{attribute 'linkalways'} 
{attribute 'no_explicit_call' := 'This FB is a CLASS and must be accessed using methods or properties'}
{attribute 'enable_dynamic_creation'}
FUNCTION_BLOCK _ETcVnFeatureScoreTypeORB EXTENDS EnumDatatypeBase
VAR
	localData : ETcVnFeatureScoreTypeORB;
	activeData : REFERENCE TO ETcVnFeatureScoreTypeORB;
	enumBaseDatatype : _DINT(localData);
END_VAR

METHOD PRIVATE AddLocalEnumeration
VAR_INPUT
	Enumeration : T_MAXSTRING;
	Value : ETcVnFeatureScoreTypeORB;
END_VAR
AddEnumeration(Enumeration, Value);
END_METHOD

PROPERTY PUBLIC Address : PVOID
GET
Address := ADR(activeData);
END_GET
END_PROPERTY

METHOD PUBLIC ClearReference
VAR_INPUT
END_VAR
activeData REF= localData;
SetBaseDatatypeReference();
END_METHOD

METHOD PUBLIC Clone : I_Datatype
VAR
    pClone : POINTER TO _ETcVnFeatureScoreTypeORB;
END_VAR
pClone := __NEW(_ETcVnFeatureScoreTypeORB(InitialValue := Value));
Clone := pClone^;
END_METHOD

METHOD FB_init : BOOL
VAR_INPUT
	bInitRetains : BOOL; // if TRUE, the retain variables are initialized (warm start / cold start)
	bInCopyCode : BOOL;  // if TRUE, the instance afterwards gets moved into the copy code (online change)
	InitialValue : ETcVnFeatureScoreTypeORB;
END_VAR
localData := InitialValue;
AddBaseDatatype(enumBaseDatatype);
ClearReference();

AddLocalEnumeration('TCVN_FST_ORB_HARRIS', ETcVnFeatureScoreTypeORB.TCVN_FST_ORB_HARRIS);
AddLocalEnumeration('TCVN_FST_ORB_FAST', ETcVnFeatureScoreTypeORB.TCVN_FST_ORB_FAST);
END_METHOD

PROPERTY PUBLIC Identifier : T_MAXSTRING
GET
Identifier := 'ETcVnFeatureScoreTypeORB';
END_GET
END_PROPERTY

METHOD IsEnumeratorValueEqual : BOOL
VAR_INPUT
	Enumerator : I_KeyValueForwardEnumerator;
END_VAR
VAR
	storedValue : ETcVnFeatureScoreTypeORB;
END_VAR
IF NOT Enumerator.TryGet(storedValue) THEN
	RETURN;
END_IF

IsEnumeratorValueEqual := storedValue = activeData;
END_METHOD

METHOD PUBLIC MakeReferenceTo
VAR_INPUT
	ReferenceTarget : REFERENCE TO ETcVnFeatureScoreTypeORB;
END_VAR
activeData REF= ReferenceTarget;
SetBaseDatatypeReference();
END_METHOD

METHOD PROTECTED SetBaseDatatypeReference
VAR_INPUT
END_VAR
enumBaseDatatype.MakeReferenceTo(activeData);
END_METHOD

PROPERTY PUBLIC Size : UDINT
GET
Size := SIZEOF(activeData);
END_GET
END_PROPERTY

METHOD TryMakeReferenceTo : BOOL
VAR_INPUT
	Target : I_Datatype;
END_VAR
VAR
	targetAsEnum : I_EnumDatatype;
	pTargetData : POINTER TO ETcVnFeatureScoreTypeORB;
END_VAR
IF NOT Target.TryResolveAsEnumDatatype(targetAsEnum) THEN
	RETURN;
END_IF

IF targetAsEnum.Identifier <> Identifier THEN
	RETURN;
END_IF

pTargetData := Target.Address;
activeData REF= pTargetData^;
SetBaseDatatypeReference();
TryMakeReferenceTo := TRUE;
END_METHOD

PROPERTY PUBLIC Value : ETcVnFeatureScoreTypeORB
GET
Value := activeData;
END_GET
SET
activeData := Value;
END_SET
END_PROPERTY

END_FUNCTION_BLOCK

(* stored: Version 1.1.0.1
   POU _ETcVnFeatureScoreTypeORB: Id {aec3f79a-901e-47e4-8eb2-ed3befca7338}, SpecialFunc None
   Folder Constructor: Id {30438420-87c2-4c20-9209-e8a703bad08b}
   Folder Private: Id {11832ee0-5c87-4f87-b7cb-e28e31e438f7}
   Folder Protected: Id {fd30cff9-8363-4c26-87a0-cbf6488896b3}
   Method AddLocalEnumeration: Id {243a19e0-f10c-4b2b-b880-9ac12c75519c}
   Property Address: Id {68294dde-63b6-4751-9e25-566b55d32ca0}
   Get Get: Id {51ebfe4b-b5eb-46e2-96bc-1e75c2bb2a54}
   Method ClearReference: Id {aab946d2-f5ad-4e26-adf8-f15b34eae3e9}
   Method Clone: Id {df9b61d6-eba8-4bf0-b1c8-83e3da4ec544}
   Method FB_init: Id {f71c27f6-fda0-4646-bcff-f5c21e303e81}
   Property Identifier: Id {e36e0c6d-10a9-4166-ae05-f158163778ea}
   Get Get: Id {1b21ba53-0ed3-46dd-83c2-39fcda666826}
   Method IsEnumeratorValueEqual: Id {9030eea2-a14a-47e6-ab5f-40867430f8af}
   Method MakeReferenceTo: Id {1ba42711-7944-4ef3-aeff-1f15248875f0}
   Method SetBaseDatatypeReference: Id {22fa8352-fd66-4982-bcc2-9dd51ed89b96}
   Property Size: Id {f077f3e3-9388-4d88-9964-223492e6d787}
   Get Get: Id {ba872d34-9798-4fc1-bfe3-e33bc0c1a2ed}
   Method TryMakeReferenceTo: Id {8a432a57-e800-4bbf-bbff-7b674e3541cb}
   Property Value: Id {46154517-e6da-4c0e-96c8-20a83d2498f9}
   Get Get: Id {08303e38-8d06-4da5-a1f0-c699609d5a34}
   Set Set: Id {9db16d59-cbad-4a5e-9bd0-32a58243f179} *)
